// TIA Portal V19 export
FUNCTION_BLOCK "TYPIC_C501_IF_NME"   // FB62, FBD
TITLE = TYPIC_C501_IF_NME: Niveaumeting
{ S7_Optimized_Access := 'TRUE' }
AUTHOR : OCOTECH
FAMILY : Typical
NAME : C501.702
// Logisch Object Besturing: C501.702
// 
// De interne functie niveaumeting verzorgt de interne besturing en bewaking van een niveaumeting van de brandblusinstallatie.
// stored: MemoryReserve 10, SetENOAutomatically false
   VAR_INPUT
      EXT_HW { ExternalAccessible := 'False'; ExternalVisible := 'False'; ExternalWritable := 'False'} : Bool;   // Sturings hardware (PLC) bewaking (1 = OK)
      IN_MWA { ExternalAccessible := 'False'; ExternalVisible := 'False'; ExternalWritable := 'False'} : Word;   // Meetwaarde
      IN_HW { ExternalAccessible := 'False'; ExternalVisible := 'False'; ExternalWritable := 'False'} : Bool;   // Vlotter: 1 = Bovenwater / 0 = Onderwater
      IN_VHW { ExternalAccessible := 'False'; ExternalVisible := 'False'; ExternalWritable := 'False'} : Bool;   // Vlotter: 1 = Bovenwater / 0 = Onderwater
      IN_SD { ExternalAccessible := 'False'; ExternalVisible := 'False'; ExternalWritable := 'False'} : Bool;   // Vlotter: 1 = Bovenwater / 0 = Onderwater
      IN_SO { ExternalAccessible := 'False'; ExternalVisible := 'False'; ExternalWritable := 'False'} : Bool;   // Vlotter: 1 = Onderwater / 0 = Bovenwater
      IN_VRL { ExternalAccessible := 'False'; ExternalVisible := 'False'; ExternalWritable := 'False'} : Bool;   // Vlotter: 1 = Onderwater / 0 = Bovenwater
      IN_RL { ExternalAccessible := 'False'; ExternalVisible := 'False'; ExternalWritable := 'False'} : Bool;   // Vlotter: 1 = Onderwater / 0 = Bovenwater
      IN_AUT_C501 { ExternalAccessible := 'False'; ExternalVisible := 'False'; ExternalWritable := 'False'} : Bool;   // Beveiligingen: serie geschakelde terugmelding (1= OK)
      CFG_MAX { ExternalAccessible := 'False'; ExternalVisible := 'False'; ExternalWritable := 'False'} : Int;   // Waarde van input IN_MWA als maximum voor de scalering ter bepaling van NIV_MWA
      CFG_MIN { ExternalAccessible := 'False'; ExternalVisible := 'False'; ExternalWritable := 'False'} : Int;   // Waarde van input IN_MWA als minimum voor de scalering ter bepaling van NIV_MWA
      CFG_MAX_SWA { ExternalAccessible := 'False'; ExternalVisible := 'False'; ExternalWritable := 'False'} : Real;   // Waarde die toegekend wordt aan NIV_MWA als maximumwmaximumwaarde voor de meeteenheid
      CFG_MIN_SWA { ExternalAccessible := 'False'; ExternalVisible := 'False'; ExternalWritable := 'False'} : Real;   // Waarde die toegekend wordt aan NIV_MWA als minimumwmaximumwaarde voor de meeteenheid
   END_VAR
   VAR_OUTPUT
      VAR_IF_NME { ExternalAccessible := 'False'; ExternalVisible := 'False'; ExternalWritable := 'False'} : "C501_VAR_IF_NME_TYPIC";   // Struct met alle variabelen naar de basisfunctie
   END_VAR
   VAR
      STO { ExternalWritable := 'False'} : Struct   // Storingen
         A001 : Bool;   // Beveiliging aangesproken
         A002 : Bool;   // Draadbreuk analoge meting
         A003 : Bool;   // Meetbereik overschreden
         A004 : Bool;   // Status vlotters inconsistent
      END_STRUCT;
      VAR { ExternalWritable := 'False'} : Struct   // Variabelen
         MWA : Real;   // Meetwaarde
         HW : USInt;   // Hoogwater vlotter
         VHW : USInt;   // Voorwaarschuwing hoogwater
         SD : USInt;   // Suppletie dicht
         SO : USInt;   // Suppletie open
         VRL : USInt;   // Voorwaarschuwing reservoir leeg
         RL : USInt;   // Reservoir leeg
         EXT_HW { ExternalAccessible := 'False'; ExternalVisible := 'False'} : Bool;   // Sturings hardware (PLC) in storing
      END_STRUCT;
   END_VAR
BEGIN

REGION Network 1: START
END_REGION

REGION Network 2: +++ Bepalen status peilen (vlotters) +++
   // Aan de hand van de status van de vlotters (inputs) wordt het peil (onderwater/bovenwater) bepaalt.
END_REGION

REGION Network 3: +++ Meting +++
   // Verwerken van de analoge meting.
END_REGION

REGION Network 4: +++ Storingen +++
   // Verwerken van de storingsmeldingen.
END_REGION

REGION Network 5: Storing A001: Beveiliging aangesproken
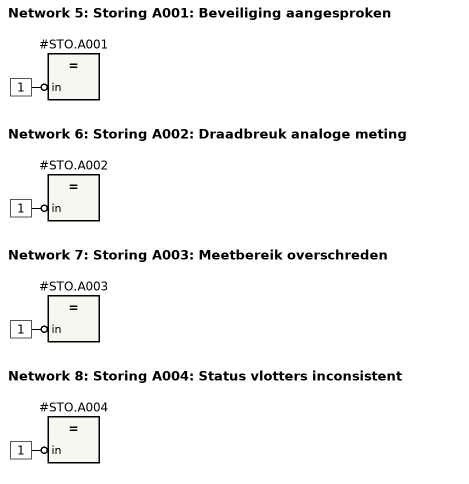
   #STO.A001 := NOT 1;
END_REGION

REGION Network 6: Storing A002: Draadbreuk analoge meting
   #STO.A002 := NOT 1;
END_REGION

REGION Network 7: Storing A003: Meetbereik overschreden
   #STO.A003 := NOT 1;
END_REGION

REGION Network 8: Storing A004: Status vlotters inconsistent
   #STO.A004 := NOT 1;
END_REGION

REGION Network 9 (SCL): EINDE
   // Variabelen van intern scada rakvlak naar outputs copieren
   #VAR_IF_NME.MWA := #VAR.MWA;
   #VAR_IF_NME.HW := #VAR.HW;
   #VAR_IF_NME.VHW := #VAR.VHW;
   #VAR_IF_NME.SD := #VAR.SD;
   #VAR_IF_NME.SO := #VAR.SO;
   #VAR_IF_NME.VRL := #VAR.VRL;
   #VAR_IF_NME.RL := #VAR.RL;
   #VAR_IF_NME.EXT_HW := #VAR.EXT_HW;
   #VAR_IF_NME.STO := #STO;
END_REGION
END_FUNCTION_BLOCK
